(* Logix 5000 project; controller cal1615 1756-L62 rev 20.19; software revision 20.05; part 55 of 81 *)
(* tags used below, declared in another part *)
   FAULT : BOOL;   // Fault AFI
   p01_param_fan_zero_speed : REAL;
   p01_param_mtr_over_speed_pct : REAL;   // System Parameter Metering Roll Overspeed [pct]
   p01_param_tension_deviation : REAL;
   p01_recipe_active : recipe;   // Active Recipe
   p01r02_plc_scan_time_in_sec : REAL;   // System PLC Scan Time in Seconds
   p01r09_pb_global_reset : BOOL;   // System Modes PB: Global Fault Reset
   p01r09_stretch_mode : BOOL;
   p01r12_master_ramped_speed : REAL;   // System Line Accel Decel Control Master Ramped Speed
   p01r13_line_running : BOOL;   // System Line Start Sequence Line Running
   p01r13_line_slow_ramp : BOOL;   // System Line Start Sequence Start Line to Slow Speed
   p01r13_permissive_drives : BOOL;   // System Line Start Sequence Permissive Drives
   p01r13_state : DINT;   // System Line Start Sequence Sequencer Step
   p02_dint_from_hmi : hmi_dint;
   p11r02_shutdown_temp : BOOL;   // Zone 1 Misc Control Safe Shutdown Temperature
   p11r30 : routine;   // Zone 1 Temperature Control
   p12r02_shutdown_temp : BOOL;   // Zone 2 Misc Control Safe Shutdown Temperature
   p12r15_mtr_roll_speed_offset : REAL;   // Impreg Metering Roll VFD Speed Offset
   p12r30 : routine;   // Zone 2 Temperature Control
   p22r01 : routine;   // Tension Stand 1 Main
   p22r10_pid_psn : PID;   // Tension Stand 1 Speed Tension PID Dancer Position
   p22r11 : routine;   // Tension Stand 1 VFD
   p23_ai_supply_rpm : REAL;   // Impreg Analog Inputs Supply Fan RPM
   p23_ao_selected_speed : REAL;   // Impreg Metering Roll VFD Selected Speed
   p23_ao_supply_selected_speed : REAL;   // Impreg Supply VFD Selected Speed
   p23_ave : CONTROL;   // Impreg Metering Roll VFD Avererage
   p23_di_filter_clean : BOOL;
   p23_di_metering_roll : acs800_di_normal;   // Impreg Digital Inputs Metering Roll VFD
   p23_di_supply : acs800_di_normal;   // Impreg Supply VFD VFD Inputs
   p23_di_supply_motor_therm : BOOL;   // Impreg Inputs Supply Fan Motor Thermostat
   p23_di_supply_speed_ok : BOOL;
   p23_di_therm : BOOL;   // Impreg Inputs Metering Roll Motor Temperature Ok
   p23_di_vfd_jog_fwd : BOOL;   // Impreg Input PB: VFD Jog FWD
   p23_di_vfd_jog_rev : BOOL;   // Impreg Input PB: VFD Jog REV
   p23_do_impreg : acs800_do_normal;   // Impreg Digital Outputs VFD
   p23_do_supply : acs800_do_normal;   // Impreg Supply VFD] Outputs
   p23_mtr_acc_rate : REAL;
   p23_mtr_decel_rate : REAL;
   p23_param_min_start_tension : REAL;
   p23_param_minus_adj_rate : REAL;
   p23_param_mtr_jog_speed : REAL;   // System Parameter Metering Roll Jog Speed
   p23_param_plus_adj_rate : REAL;
   p23r01 : routine;   // Impreg Main
   p23r02 : routine;   // Impreg Misc Control
   p23r09_mode_run : BOOL;   // Impreg Modes Pick Up Roll Run Mode
   p23r13 : routine;
   p23r13_pb_start : BOOL;   // Impreg Supply VFD Start
   p23r13_pb_stop : BOOL;   // Impreg Supply VFD Stop
   p23r13_request_auto_run : BOOL;   // Impreg Supply Fan VFD Request Auto Run
   p23r13_run_permissive : BOOL;   // Impreg Supply VFD Run Permissive
   p23r13_timer_fault : TIMER[10];   // Impreg Supply VFD Fault Dwell Timer
   p23r13_timer_warning : TIMER[4];   // Impreg Supply VFD Warning Dwell Timer
   p23r13_vfd_stopped : BOOL;   // Impreg Supply VFD Stopped
   p23r15 : routine;   // Impreg Metering Roll VFD
   p23r15_acc_decel_ramp : SYS_ACC_DEC_RAMP;   // Impreg Metering Roll VFD Accel/Decel Ramp
   p23r15_adjust_dwell1 : TIMER;   // Impreg Metering Roll VFD Adjustment Dwell Timer
   p23r15_average_tension : REAL;   // Impreg Metering Roll VFD Average Tension
   p23r15_dead_band_minus : REAL;   // Impreg Metering Roll VFD Dead Band -
   p23r15_dead_band_plus : REAL;   // Impreg Metering Roll VFD Dead Band +
   p23r15_dead_band_setpoint : REAL;
   p23r15_debounce_timer : TIMER;   // Impreg Metering Roll VFD Tension Ok Debounce Timer
   p23r15_ffl : CONTROL;   // Impreg Metering Roll VFD Avererage FFL
   p23r15_ffu_temp : REAL;
   p23r15_fll_stack : REAL[50];
   p23r15_mean_adjust_acitve : BOOL;   // Impreg Metering Roll VFD Mean Adjust Active
   p23r15_minus_adjust : REAL;
   p23r15_minus_adjust_acitve : BOOL;   // Impreg Metering Roll VFD Minus Adjust Active
   p23r15_minus_offset : REAL;
   p23r15_neutral_offset : REAL;
   p23r15_permissive_jog : BOOL;   // Impreg Impreg VFD Permissive Jog
   p23r15_permissive_run : BOOL;   // Impreg Metering Roll VFD Permissive Run
   p23r15_plus_adjust : REAL;
   p23r15_plus_adjust_acitve : BOOL;   // Impreg Plus Adjust Active
   p23r15_plus_offset : REAL;
   p23r15_request_jog_fwd : BOOL;   // Impreg Metering Roll VFD Request Jog FWD
   p23r15_request_jog_rev : BOOL;   // Impreg Metering Roll VFD Request Jog REV
   p23r15_request_line_run : BOOL;   // Impreg Metering Roll VFD Request Line Run
   p23r15_request_thread_fwd : BOOL;   // Impreg Metering Roll VFD Request Thread FWD
   p23r15_request_thread_rev : BOOL;   // Impreg Metering Roll VFD Request Thread REV
   p23r15_sample_timer : TIMER;   // Impreg Metering Roll Sample Timer
   p23r15_selected_speed : REAL;   // Impreg Metering Roll VFD Selected Speed
   p23r15_timer_fault : TIMER[10];   // Impreg Pick Up Roll VFD Fault Timer
   p23r15_timer_warning : TIMER[5];   // Impreg Pick Up Roll VFD Warning Timer
   p23r15_ts1_tension_ok : BOOL;   // Impreg Metering Roll VFD TS 1 Tension Ok
   p23r15_zero_speed : BOOL;   // Impreg Metering Roll VFD At Zero Speed
   p25_ai_ts2_lc : REAL;   // System Metering Roll VFD Minimum Start Tension
   p25r11_request_thread_fwd : BOOL;   // Tension Stand 2 VFD Request Thread FWD
   p25r11_request_thread_rev : BOOL;   // Tension Stand 2 VFD Request Thread REV
(* P23_Impreg, continued *)

ROUTINE R13_Supply_Fan_VFD   (* ladder *)
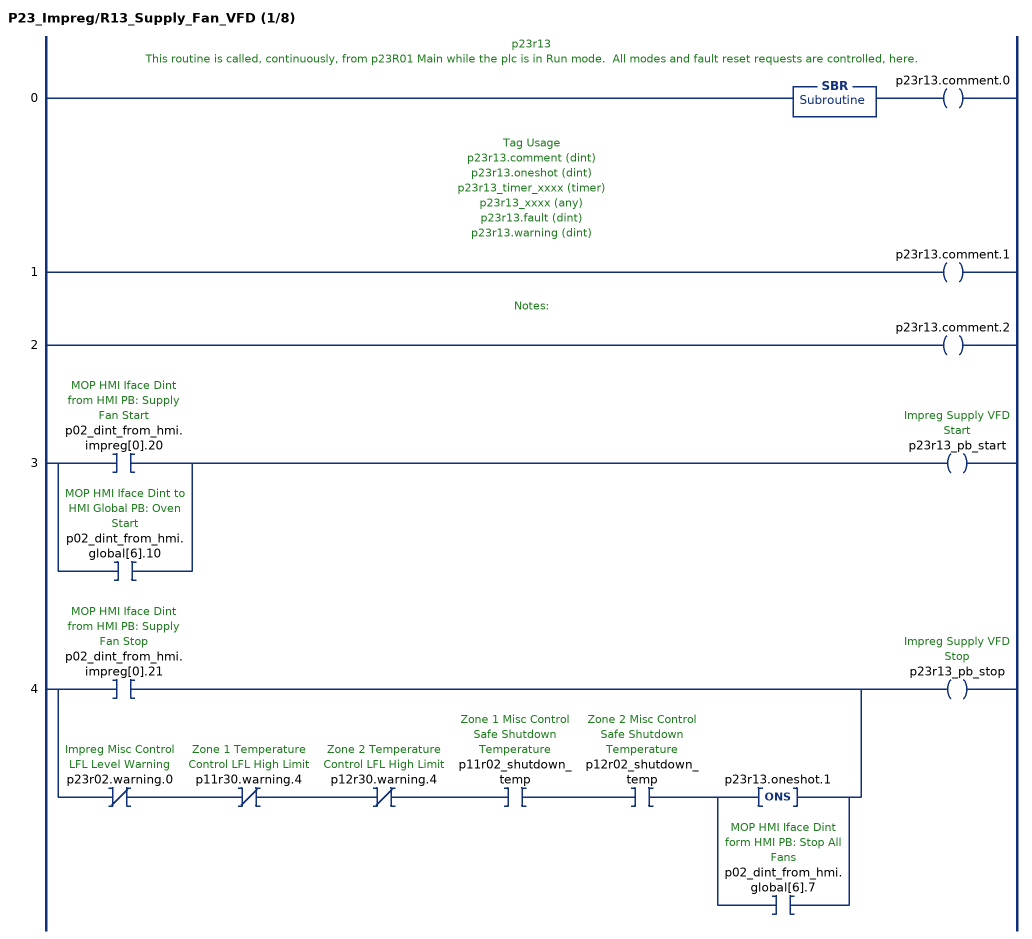
   // p23r13
   // This routine is called, continuously, from p23R01 Main while the plc is in Run mode.  All modes and fault reset requests are controlled, here.
   0: SBR()OTE(p23r13.comment.0);
   // Tag Usage
   // p23r13.comment (dint)
   // p23r13.oneshot (dint)
   // p23r13_timer_xxxx (timer)
   // p23r13_xxxx (any)
   // p23r13.fault (dint)
   // p23r13.warning (dint)
   1: OTE(p23r13.comment.1);
   // Notes:
   2: OTE(p23r13.comment.2);
   3: [XIC(p02_dint_from_hmi.impreg[0].20) ,XIC(p02_dint_from_hmi.global[6].10) ]OTE(p23r13_pb_start);
   4: [XIC(p02_dint_from_hmi.impreg[0].21) ,XIO(p23r02.warning.0) XIO(p11r30.warning.4) XIO(p12r30.warning.4) XIC(p11r02_shutdown_temp) XIC(p12r02_shutdown_temp) [ONS(p23r13.oneshot.1) ,XIC(p02_dint_from_hmi.global[6].7) ] ]OTE(p23r13_pb_stop);
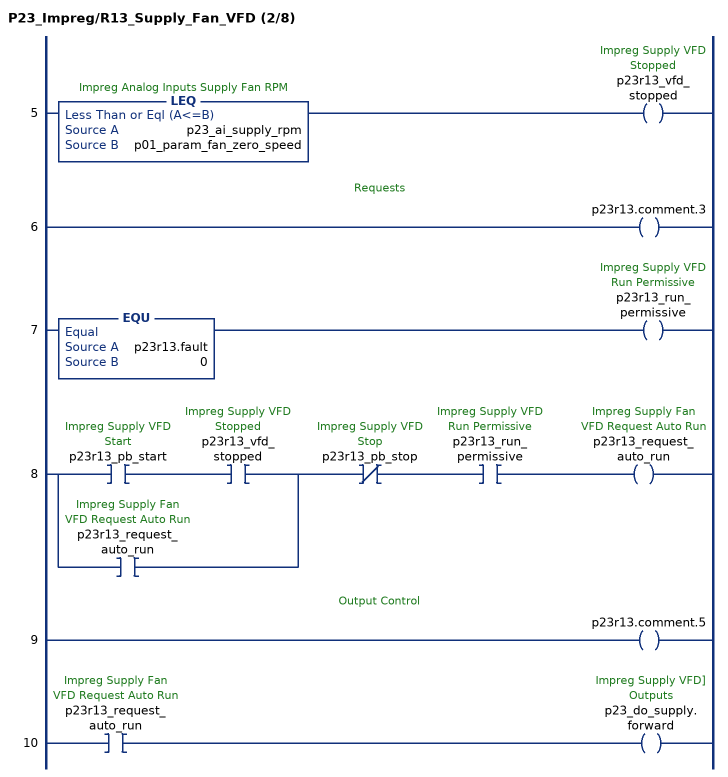
   5: LEQ(p23_ai_supply_rpm,p01_param_fan_zero_speed)OTE(p23r13_vfd_stopped);
   // Requests
   6: OTE(p23r13.comment.3);
   7: EQU(p23r13.fault,0)OTE(p23r13_run_permissive);
   8: [XIC(p23r13_pb_start) XIC(p23r13_vfd_stopped) ,XIC(p23r13_request_auto_run) ]XIO(p23r13_pb_stop)XIC(p23r13_run_permissive)OTE(p23r13_request_auto_run);
   // Output Control
   9: OTE(p23r13.comment.5);
   10: XIC(p23r13_request_auto_run)OTE(p23_do_supply.forward);
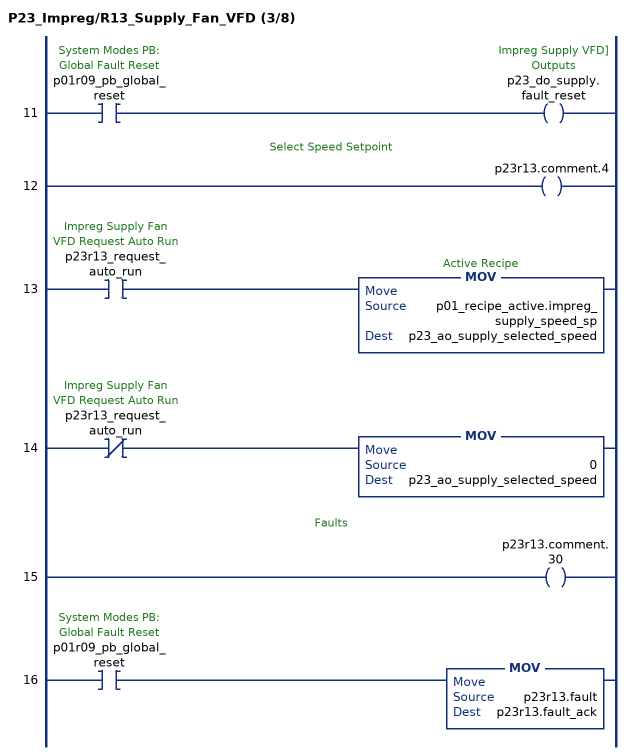
   11: XIC(p01r09_pb_global_reset)OTE(p23_do_supply.fault_reset);
   // Select Speed Setpoint
   12: OTE(p23r13.comment.4);
   13: XIC(p23r13_request_auto_run)MOV(p01_recipe_active.impreg_supply_speed_sp,p23_ao_supply_selected_speed);
   14: XIO(p23r13_request_auto_run)MOV(0,p23_ao_supply_selected_speed);
   // Faults
   15: OTE(p23r13.comment.30);
   16: XIC(p01r09_pb_global_reset)MOV(p23r13.fault,p23r13.fault_ack);
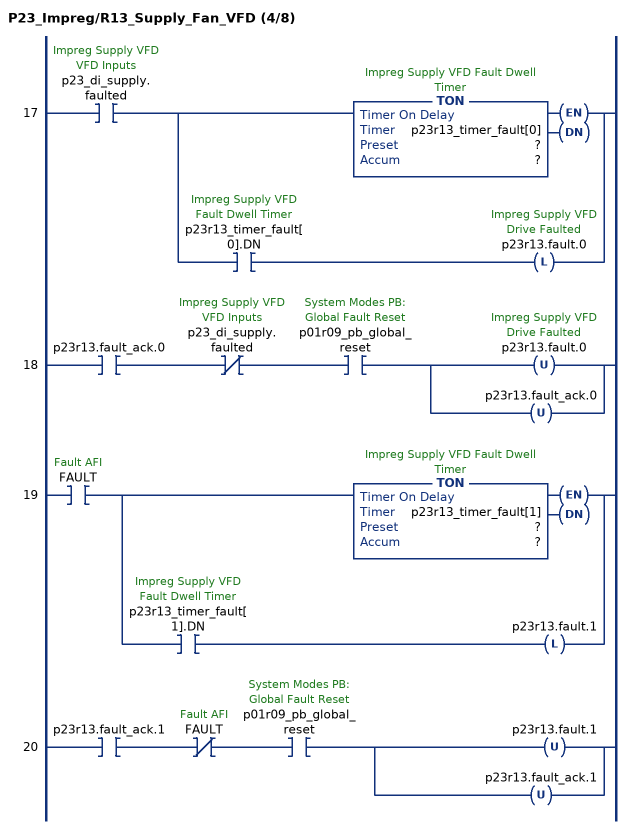
   17: XIC(p23_di_supply.faulted)[TON(p23r13_timer_fault[0],?,?) ,XIC(p23r13_timer_fault[0].DN) OTL(p23r13.fault.0) ];
   18: XIC(p23r13.fault_ack.0)XIO(p23_di_supply.faulted)XIC(p01r09_pb_global_reset)[OTU(p23r13.fault.0) ,OTU(p23r13.fault_ack.0) ];
   19: XIC(FAULT)[TON(p23r13_timer_fault[1],?,?) ,XIC(p23r13_timer_fault[1].DN) OTL(p23r13.fault.1) ];
   20: XIC(p23r13.fault_ack.1)XIO(FAULT)XIC(p01r09_pb_global_reset)[OTU(p23r13.fault.1) ,OTU(p23r13.fault_ack.1) ];
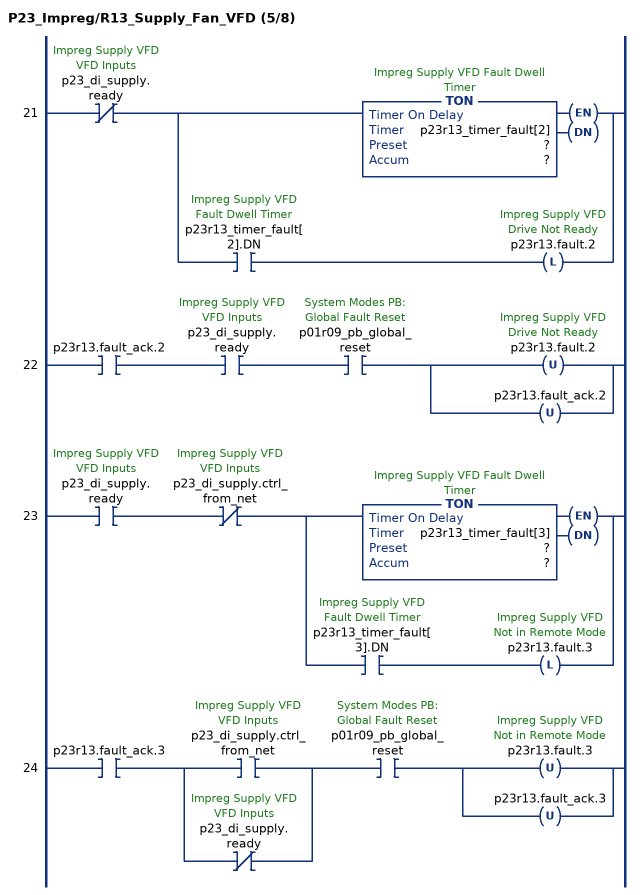
   21: XIO(p23_di_supply.ready)[TON(p23r13_timer_fault[2],?,?) ,XIC(p23r13_timer_fault[2].DN) OTL(p23r13.fault.2) ];
   22: XIC(p23r13.fault_ack.2)XIC(p23_di_supply.ready)XIC(p01r09_pb_global_reset)[OTU(p23r13.fault.2) ,OTU(p23r13.fault_ack.2) ];
   23: XIC(p23_di_supply.ready)XIO(p23_di_supply.ctrl_from_net)[TON(p23r13_timer_fault[3],?,?) ,XIC(p23r13_timer_fault[3].DN) OTL(p23r13.fault.3) ];
   24: XIC(p23r13.fault_ack.3)[XIC(p23_di_supply.ctrl_from_net) ,XIO(p23_di_supply.ready) ]XIC(p01r09_pb_global_reset)[OTU(p23r13.fault.3) ,OTU(p23r13.fault_ack.3) ];
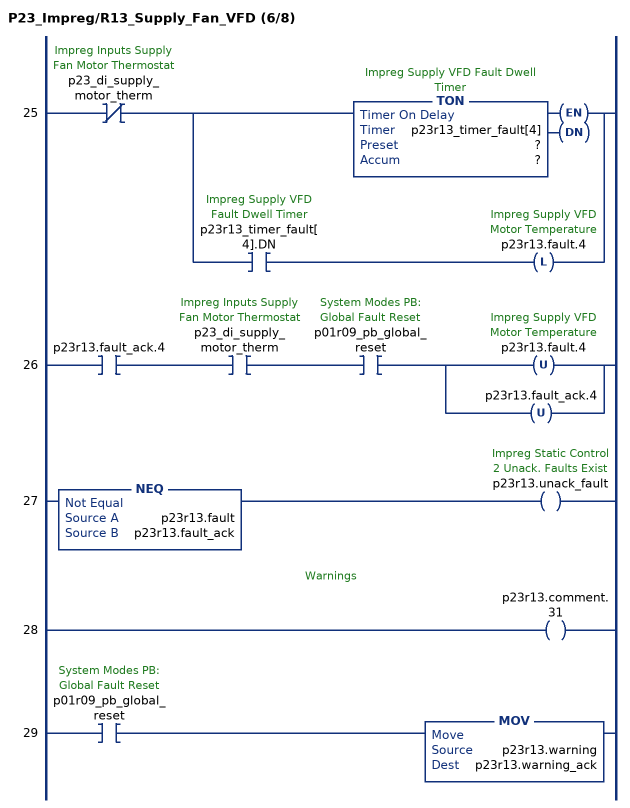
   25: XIO(p23_di_supply_motor_therm)[TON(p23r13_timer_fault[4],?,?) ,XIC(p23r13_timer_fault[4].DN) OTL(p23r13.fault.4) ];
   26: XIC(p23r13.fault_ack.4)XIC(p23_di_supply_motor_therm)XIC(p01r09_pb_global_reset)[OTU(p23r13.fault.4) ,OTU(p23r13.fault_ack.4) ];
   27: NEQ(p23r13.fault,p23r13.fault_ack)OTE(p23r13.unack_fault);
   // Warnings
   28: OTE(p23r13.comment.31);
   29: XIC(p01r09_pb_global_reset)MOV(p23r13.warning,p23r13.warning_ack);
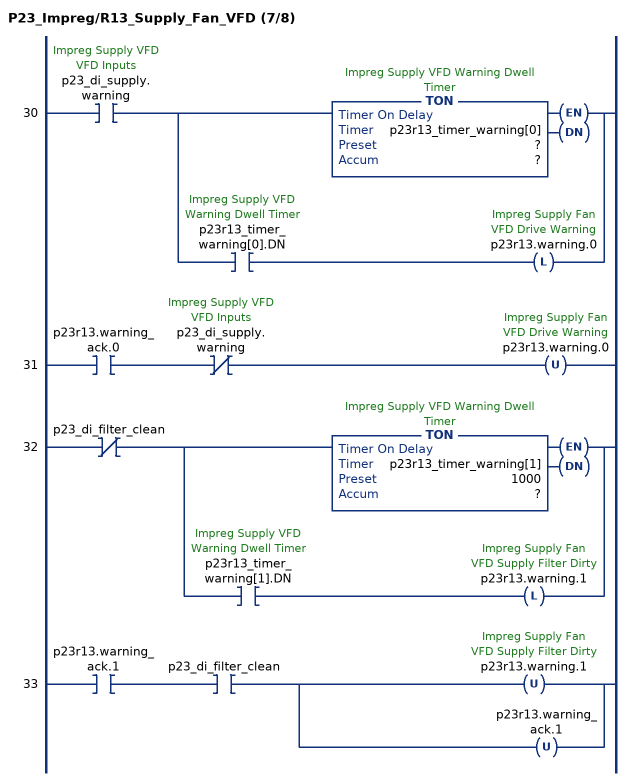
   30: XIC(p23_di_supply.warning)[TON(p23r13_timer_warning[0],?,?) ,XIC(p23r13_timer_warning[0].DN) OTL(p23r13.warning.0) ];
   31: XIC(p23r13.warning_ack.0)XIO(p23_di_supply.warning)OTU(p23r13.warning.0);
   32: XIO(p23_di_filter_clean)[TON(p23r13_timer_warning[1],?,?) ,XIC(p23r13_timer_warning[1].DN) OTL(p23r13.warning.1) ];
   33: XIC(p23r13.warning_ack.1)XIC(p23_di_filter_clean)[OTU(p23r13.warning.1) ,OTU(p23r13.warning_ack.1) ];
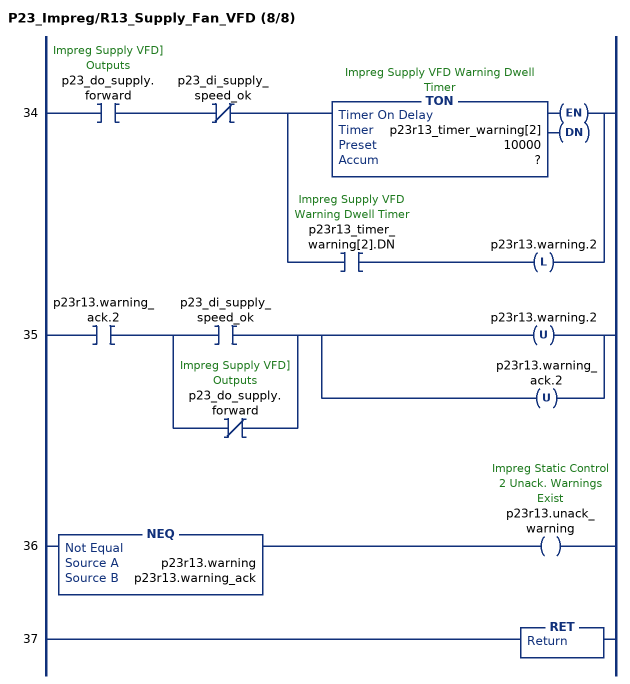
   34: XIC(p23_do_supply.forward)XIO(p23_di_supply_speed_ok)[TON(p23r13_timer_warning[2],?,?) ,XIC(p23r13_timer_warning[2].DN) OTL(p23r13.warning.2) ];
   35: XIC(p23r13.warning_ack.2)[XIC(p23_di_supply_speed_ok) ,XIO(p23_do_supply.forward) ][OTU(p23r13.warning.2) ,OTU(p23r13.warning_ack.2) ];
   36: NEQ(p23r13.warning,p23r13.warning_ack)OTE(p23r13.unack_warning);
   37: RET();
END_ROUTINE

ROUTINE R15_Metering_Roll_VFD   (* ladder *)
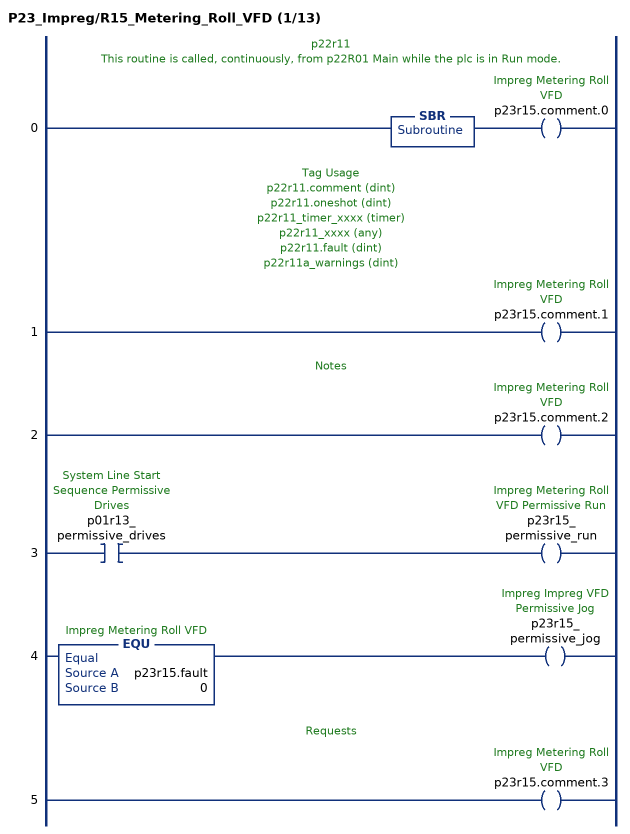
   // p22r11
   // This routine is called, continuously, from p22R01 Main while the plc is in Run mode.
   0: SBR()OTE(p23r15.comment.0);
   // Tag Usage
   // p22r11.comment (dint)
   // p22r11.oneshot (dint)
   // p22r11_timer_xxxx (timer)
   // p22r11_xxxx (any)
   // p22r11.fault (dint)
   // p22r11a_warnings (dint)
   1: OTE(p23r15.comment.1);
   // Notes
   2: OTE(p23r15.comment.2);
   3: XIC(p01r13_permissive_drives)OTE(p23r15_permissive_run);
   4: EQU(p23r15.fault,0)OTE(p23r15_permissive_jog);
   // Requests
   5: OTE(p23r15.comment.3);
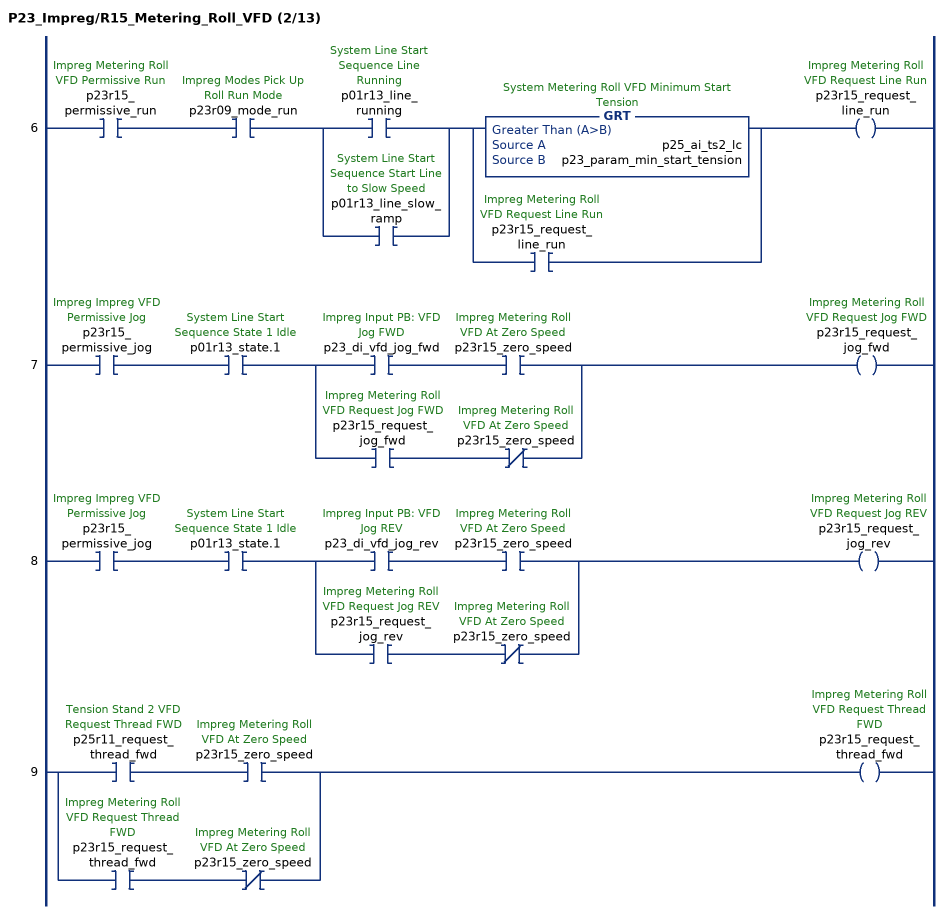
   6: XIC(p23r15_permissive_run)XIC(p23r09_mode_run)[XIC(p01r13_line_running) ,XIC(p01r13_line_slow_ramp) ][GRT(p25_ai_ts2_lc,p23_param_min_start_tension) ,XIC(p23r15_request_line_run) ]OTE(p23r15_request_line_run);
   7: XIC(p23r15_permissive_jog)XIC(p01r13_state.1)[XIC(p23_di_vfd_jog_fwd) XIC(p23r15_zero_speed) ,XIC(p23r15_request_jog_fwd) XIO(p23r15_zero_speed) ]OTE(p23r15_request_jog_fwd);
   8: XIC(p23r15_permissive_jog)XIC(p01r13_state.1)[XIC(p23_di_vfd_jog_rev) XIC(p23r15_zero_speed) ,XIC(p23r15_request_jog_rev) XIO(p23r15_zero_speed) ]OTE(p23r15_request_jog_rev);
   9: [XIC(p25r11_request_thread_fwd) XIC(p23r15_zero_speed) ,XIC(p23r15_request_thread_fwd) XIO(p23r15_zero_speed) ]OTE(p23r15_request_thread_fwd);
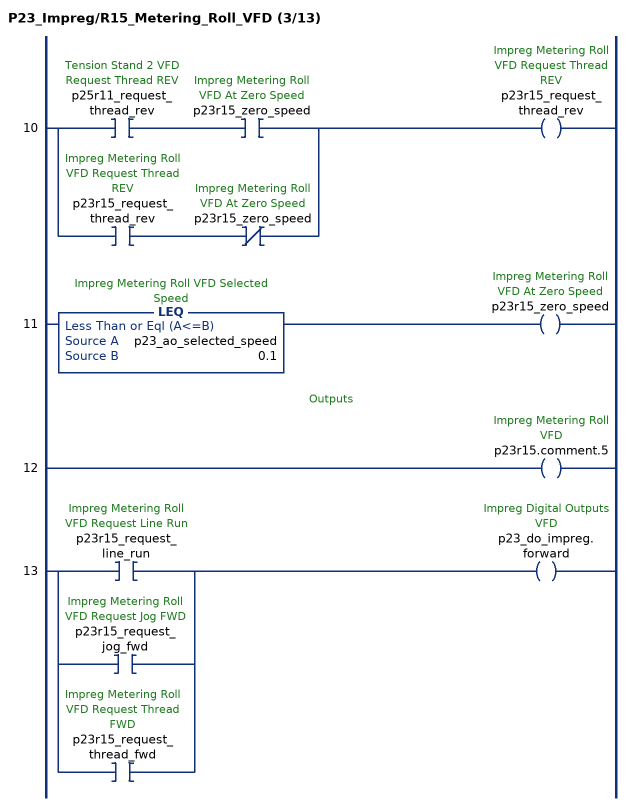
   10: [XIC(p25r11_request_thread_rev) XIC(p23r15_zero_speed) ,XIC(p23r15_request_thread_rev) XIO(p23r15_zero_speed) ]OTE(p23r15_request_thread_rev);
   11: LEQ(p23_ao_selected_speed,0.1)OTE(p23r15_zero_speed);
   // Outputs
   12: OTE(p23r15.comment.5);
   13: [XIC(p23r15_request_line_run) ,XIC(p23r15_request_jog_fwd) ,XIC(p23r15_request_thread_fwd) ]OTE(p23_do_impreg.forward);
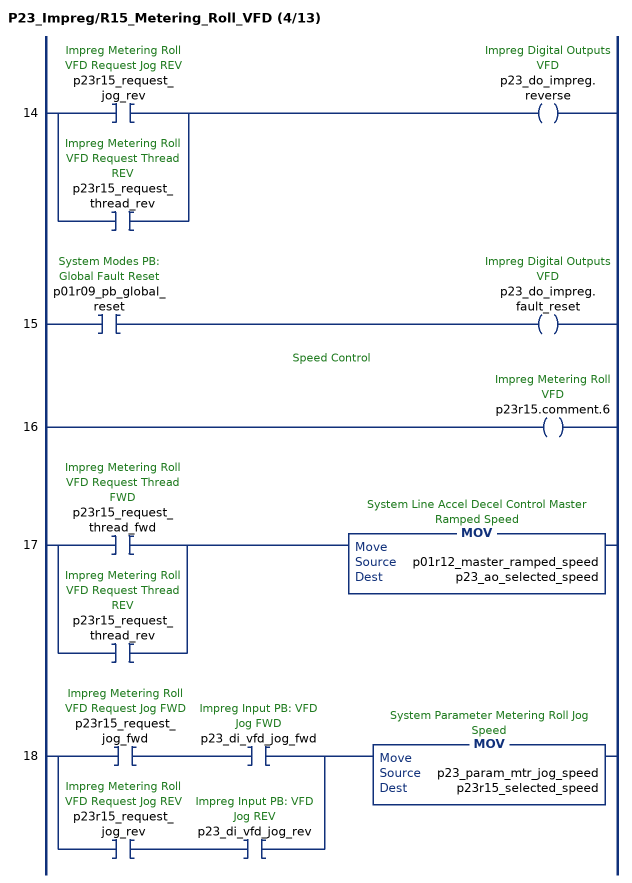
   14: [XIC(p23r15_request_jog_rev) ,XIC(p23r15_request_thread_rev) ]OTE(p23_do_impreg.reverse);
   15: XIC(p01r09_pb_global_reset)OTE(p23_do_impreg.fault_reset);
   // Speed Control
   16: OTE(p23r15.comment.6);
   17: [XIC(p23r15_request_thread_fwd) ,XIC(p23r15_request_thread_rev) ]MOV(p01r12_master_ramped_speed,p23_ao_selected_speed);
   18: [XIC(p23r15_request_jog_fwd) XIC(p23_di_vfd_jog_fwd) ,XIC(p23r15_request_jog_rev) XIC(p23_di_vfd_jog_rev) ]MOV(p23_param_mtr_jog_speed,p23r15_selected_speed);
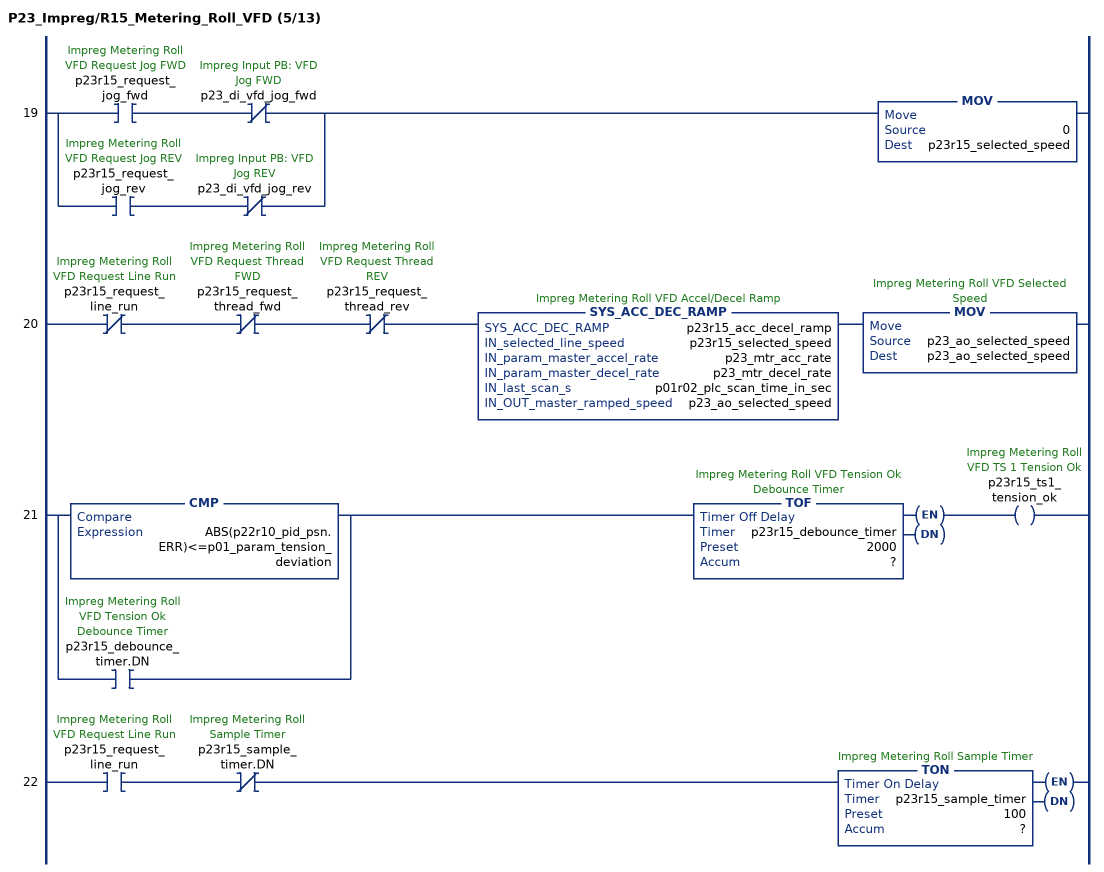
   19: [XIC(p23r15_request_jog_fwd) XIO(p23_di_vfd_jog_fwd) ,XIC(p23r15_request_jog_rev) XIO(p23_di_vfd_jog_rev) ]MOV(0,p23r15_selected_speed);
   20: XIO(p23r15_request_line_run)XIO(p23r15_request_thread_fwd)XIO(p23r15_request_thread_rev)SYS_ACC_DEC_RAMP(p23r15_acc_decel_ramp,p23r15_selected_speed,p23_mtr_acc_rate,p23_mtr_decel_rate,p01r02_plc_scan_time_in_sec,p23_ao_selected_speed)MOV(p23_ao_selected_speed,p23_ao_selected_speed);
   21: [CMP(ABS(p22r10_pid_psn.ERR)<=p01_param_tension_deviation) ,XIC(p23r15_debounce_timer.DN) ]TOF(p23r15_debounce_timer,?,?)OTE(p23r15_ts1_tension_ok);
   22: XIC(p23r15_request_line_run)XIO(p23r15_sample_timer.DN)TON(p23r15_sample_timer,?,?);
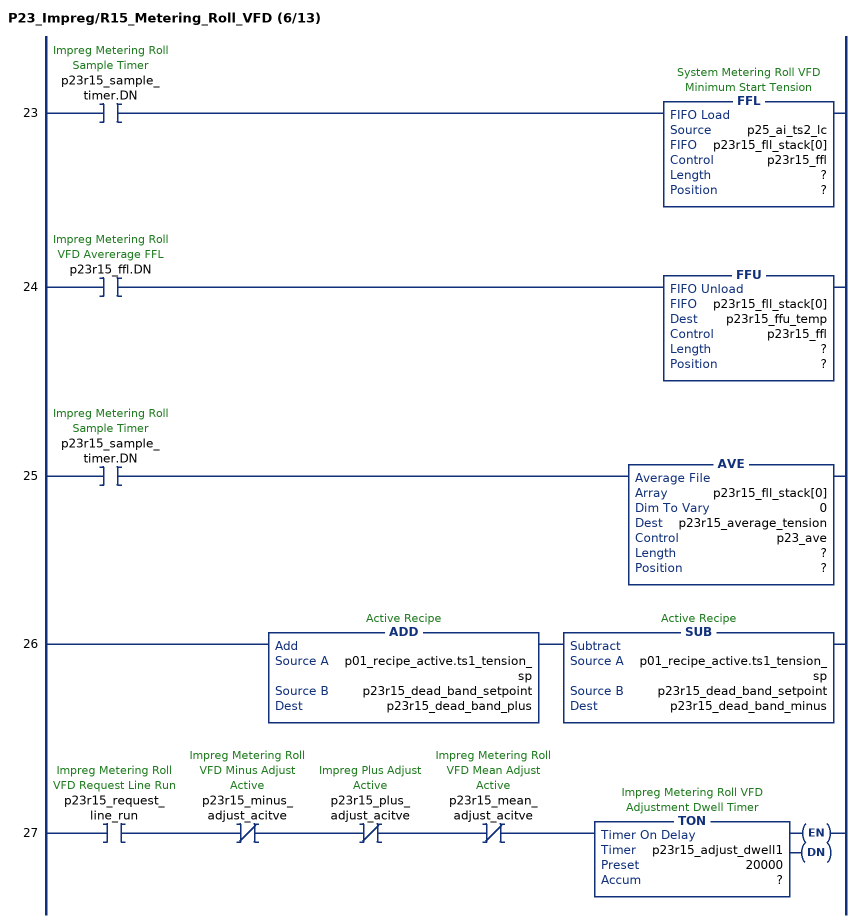
   23: XIC(p23r15_sample_timer.DN)FFL(p25_ai_ts2_lc,p23r15_fll_stack[0],p23r15_ffl,?,?);
   24: XIC(p23r15_ffl.DN)FFU(p23r15_fll_stack[0],p23r15_ffu_temp,p23r15_ffl,?,?);
   25: XIC(p23r15_sample_timer.DN)AVE(p23r15_fll_stack[0],0,p23r15_average_tension,p23_ave,?,?);
   26: ADD(p01_recipe_active.ts1_tension_sp,p23r15_dead_band_setpoint,p23r15_dead_band_plus)SUB(p01_recipe_active.ts1_tension_sp,p23r15_dead_band_setpoint,p23r15_dead_band_minus);
   27: XIC(p23r15_request_line_run)XIO(p23r15_minus_adjust_acitve)XIO(p23r15_plus_adjust_acitve)XIO(p23r15_mean_adjust_acitve)TON(p23r15_adjust_dwell1,?,?);
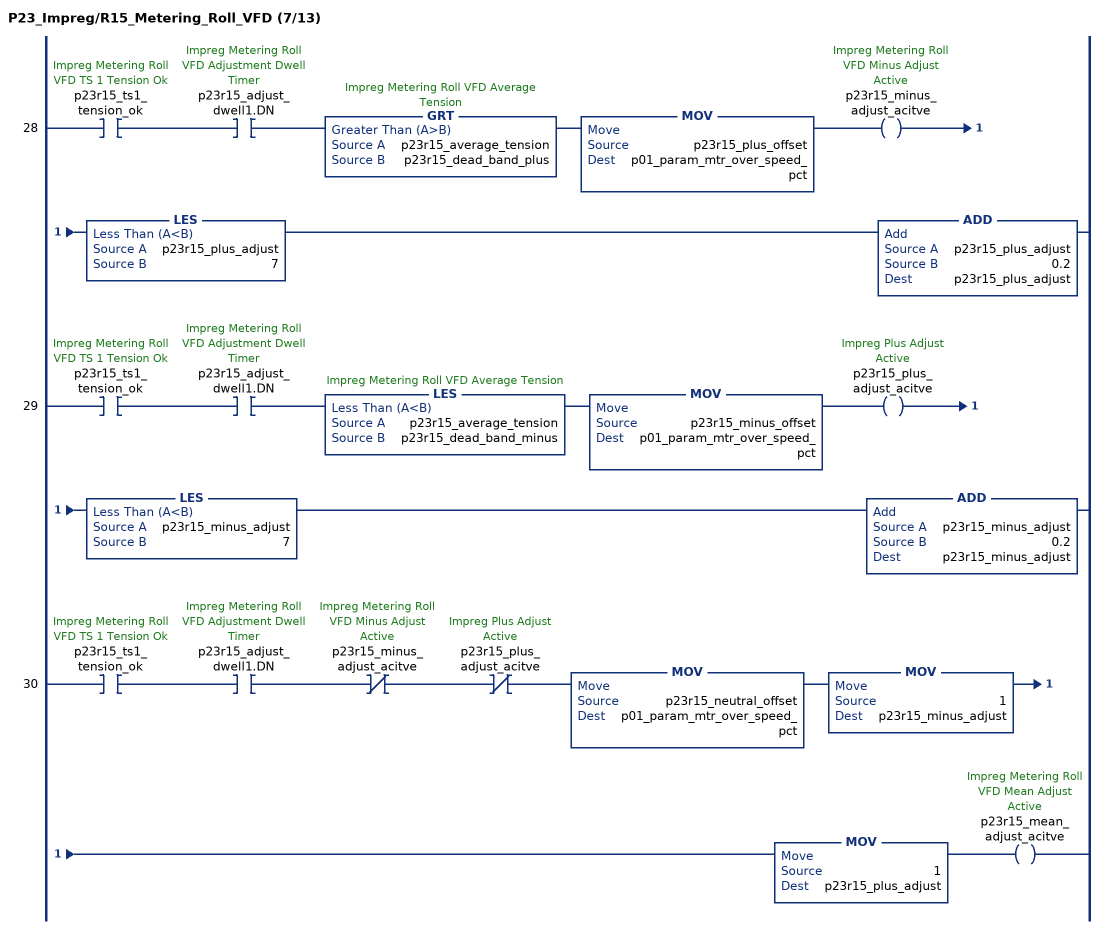
   28: XIC(p23r15_ts1_tension_ok)XIC(p23r15_adjust_dwell1.DN)GRT(p23r15_average_tension,p23r15_dead_band_plus)MOV(p23r15_plus_offset,p01_param_mtr_over_speed_pct)OTE(p23r15_minus_adjust_acitve)LES(p23r15_plus_adjust,7)ADD(p23r15_plus_adjust,0.2,p23r15_plus_adjust);
   29: XIC(p23r15_ts1_tension_ok)XIC(p23r15_adjust_dwell1.DN)LES(p23r15_average_tension,p23r15_dead_band_minus)MOV(p23r15_minus_offset,p01_param_mtr_over_speed_pct)OTE(p23r15_plus_adjust_acitve)LES(p23r15_minus_adjust,7)ADD(p23r15_minus_adjust,0.2,p23r15_minus_adjust);
   30: XIC(p23r15_ts1_tension_ok)XIC(p23r15_adjust_dwell1.DN)XIO(p23r15_minus_adjust_acitve)XIO(p23r15_plus_adjust_acitve)MOV(p23r15_neutral_offset,p01_param_mtr_over_speed_pct)MOV(1,p23r15_minus_adjust)MOV(1,p23r15_plus_adjust)OTE(p23r15_mean_adjust_acitve);
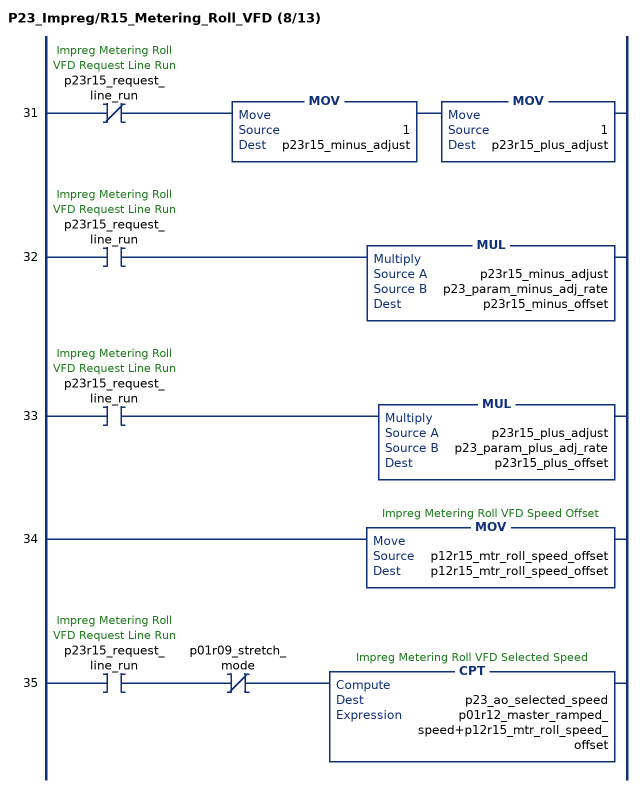
   31: XIO(p23r15_request_line_run)MOV(1,p23r15_minus_adjust)MOV(1,p23r15_plus_adjust);
   32: XIC(p23r15_request_line_run)MUL(p23r15_minus_adjust,p23_param_minus_adj_rate,p23r15_minus_offset);
   33: XIC(p23r15_request_line_run)MUL(p23r15_plus_adjust,p23_param_plus_adj_rate,p23r15_plus_offset);
   34: MOV(p12r15_mtr_roll_speed_offset,p12r15_mtr_roll_speed_offset);
   35: XIC(p23r15_request_line_run)XIO(p01r09_stretch_mode)CPT(p23_ao_selected_speed,p01r12_master_ramped_speed+p12r15_mtr_roll_speed_offset);
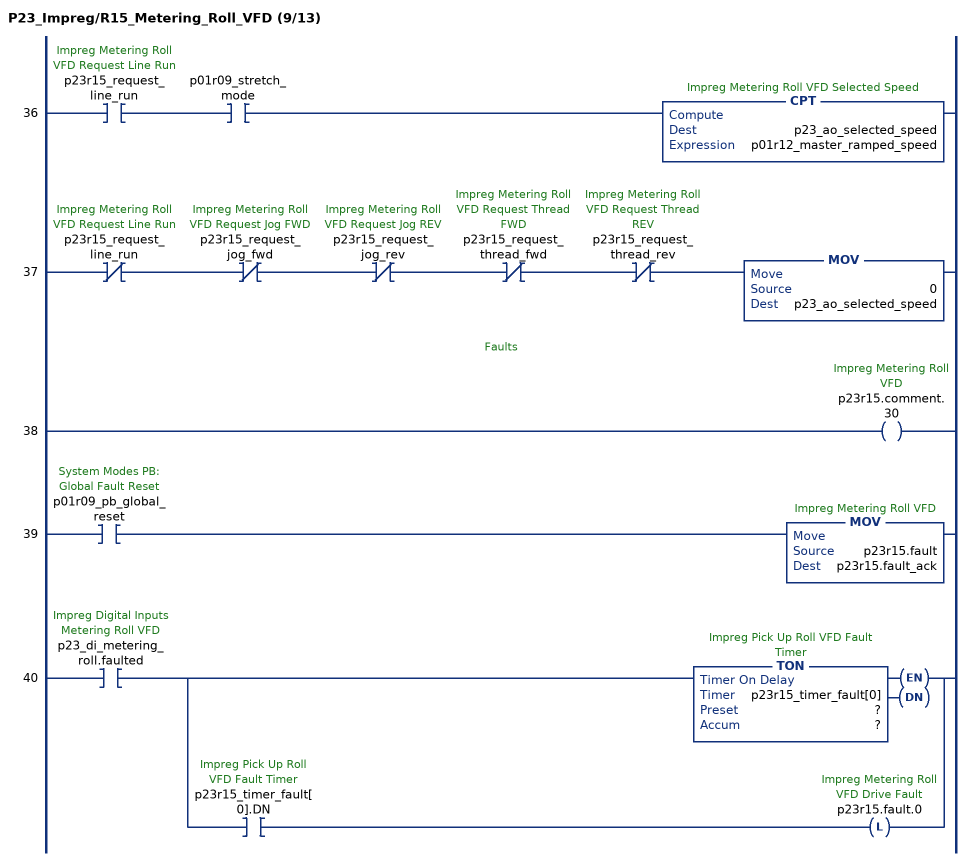
   36: XIC(p23r15_request_line_run)XIC(p01r09_stretch_mode)CPT(p23_ao_selected_speed,p01r12_master_ramped_speed);
   37: XIO(p23r15_request_line_run)XIO(p23r15_request_jog_fwd)XIO(p23r15_request_jog_rev)XIO(p23r15_request_thread_fwd)XIO(p23r15_request_thread_rev)MOV(0,p23_ao_selected_speed);
   // Faults
   38: OTE(p23r15.comment.30);
   39: XIC(p01r09_pb_global_reset)MOV(p23r15.fault,p23r15.fault_ack);
   40: XIC(p23_di_metering_roll.faulted)[TON(p23r15_timer_fault[0],?,?) ,XIC(p23r15_timer_fault[0].DN) OTL(p23r15.fault.0) ];
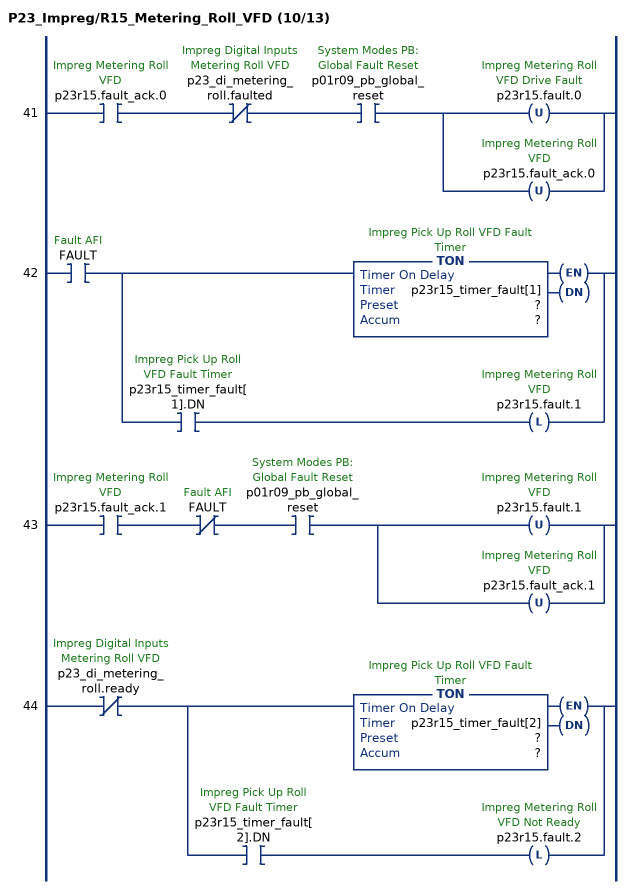
   41: XIC(p23r15.fault_ack.0)XIO(p23_di_metering_roll.faulted)XIC(p01r09_pb_global_reset)[OTU(p23r15.fault.0) ,OTU(p23r15.fault_ack.0) ];
   42: XIC(FAULT)[TON(p23r15_timer_fault[1],?,?) ,XIC(p23r15_timer_fault[1].DN) OTL(p23r15.fault.1) ];
   43: XIC(p23r15.fault_ack.1)XIO(FAULT)XIC(p01r09_pb_global_reset)[OTU(p23r15.fault.1) ,OTU(p23r15.fault_ack.1) ];
   44: XIO(p23_di_metering_roll.ready)[TON(p23r15_timer_fault[2],?,?) ,XIC(p23r15_timer_fault[2].DN) OTL(p23r15.fault.2) ];
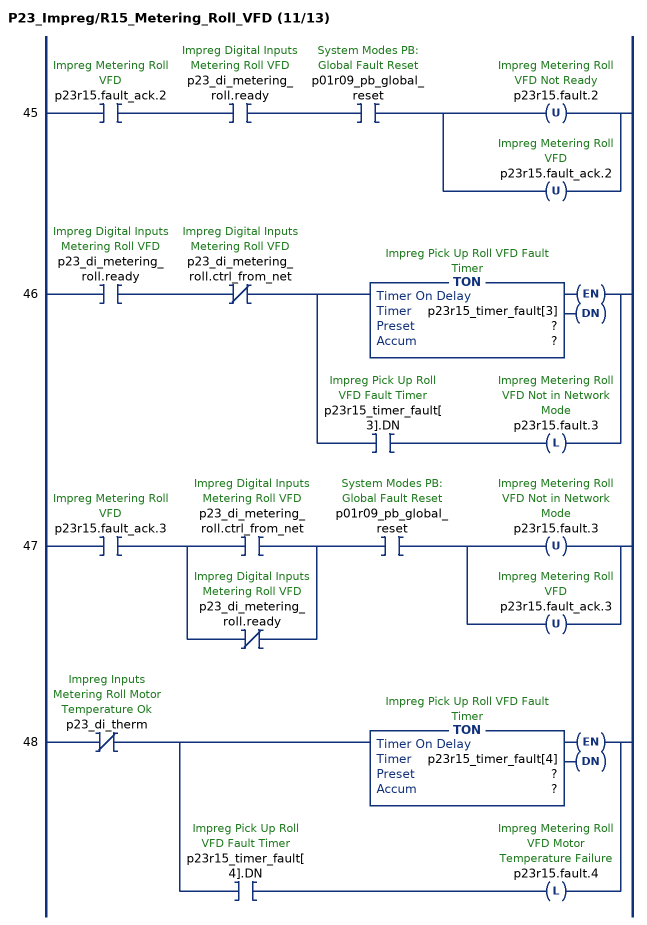
   45: XIC(p23r15.fault_ack.2)XIC(p23_di_metering_roll.ready)XIC(p01r09_pb_global_reset)[OTU(p23r15.fault.2) ,OTU(p23r15.fault_ack.2) ];
   46: XIC(p23_di_metering_roll.ready)XIO(p23_di_metering_roll.ctrl_from_net)[TON(p23r15_timer_fault[3],?,?) ,XIC(p23r15_timer_fault[3].DN) OTL(p23r15.fault.3) ];
   47: XIC(p23r15.fault_ack.3)[XIC(p23_di_metering_roll.ctrl_from_net) ,XIO(p23_di_metering_roll.ready) ]XIC(p01r09_pb_global_reset)[OTU(p23r15.fault.3) ,OTU(p23r15.fault_ack.3) ];
   48: XIO(p23_di_therm)[TON(p23r15_timer_fault[4],?,?) ,XIC(p23r15_timer_fault[4].DN) OTL(p23r15.fault.4) ];
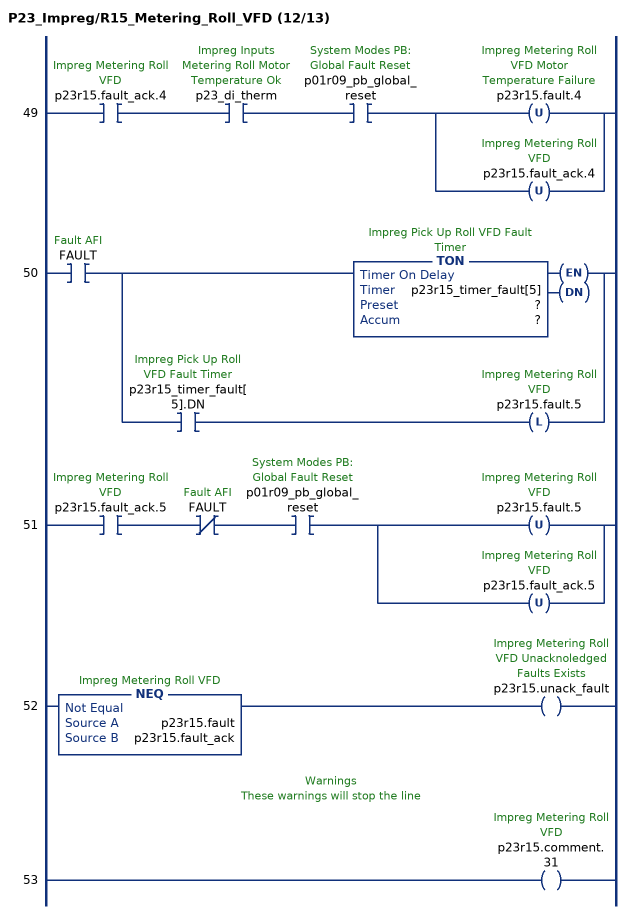
   49: XIC(p23r15.fault_ack.4)XIC(p23_di_therm)XIC(p01r09_pb_global_reset)[OTU(p23r15.fault.4) ,OTU(p23r15.fault_ack.4) ];
   50: XIC(FAULT)[TON(p23r15_timer_fault[5],?,?) ,XIC(p23r15_timer_fault[5].DN) OTL(p23r15.fault.5) ];
   51: XIC(p23r15.fault_ack.5)XIO(FAULT)XIC(p01r09_pb_global_reset)[OTU(p23r15.fault.5) ,OTU(p23r15.fault_ack.5) ];
   52: NEQ(p23r15.fault,p23r15.fault_ack)OTE(p23r15.unack_fault);
   // Warnings
   // These warnings will stop the line
   53: OTE(p23r15.comment.31);
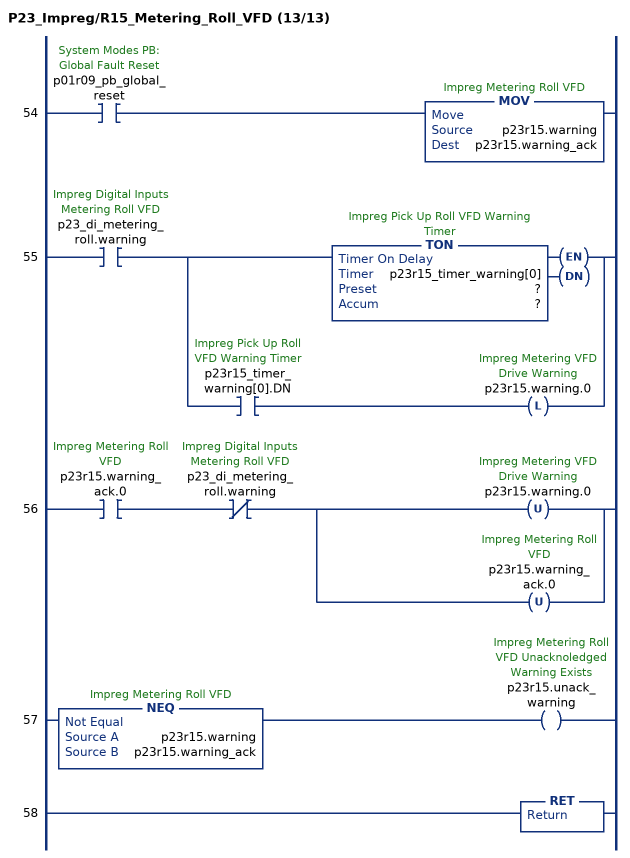
   54: XIC(p01r09_pb_global_reset)MOV(p23r15.warning,p23r15.warning_ack);
   55: XIC(p23_di_metering_roll.warning)[TON(p23r15_timer_warning[0],?,?) ,XIC(p23r15_timer_warning[0].DN) OTL(p23r15.warning.0) ];
   56: XIC(p23r15.warning_ack.0)XIO(p23_di_metering_roll.warning)[OTU(p23r15.warning.0) ,OTU(p23r15.warning_ack.0) ];
   57: NEQ(p23r15.warning,p23r15.warning_ack)OTE(p23r15.unack_warning);
   58: RET();
END_ROUTINE
